SUBAPPLICATION Uebung_230 (* Analog-Eingang *)
  (* Standard: 61499-2; Description: Copyright (c) 2023 Meisterschulen am Ostbahnhof This program and the accompanying materials are made available under the terms of the Eclipse Public License 2.0 which is available at https://www.eclipse.org/legal/epl-2.0/ SPDX-License-Identifier: EPL-2.0 *)
  (* Version 1.0, 2023-10-23, Franz Höpfinger, Meisterschulen am Ostbahnhof, initial API and implementation and/or initial documentation *)
  PACKAGE Uebungen;
  IMPORT DataPanel::io::MI::AI::DataPanel_MI_AI::AnalogInput_1A;
  IMPORT DataPanel::io::MI::const::MI::MI_00;
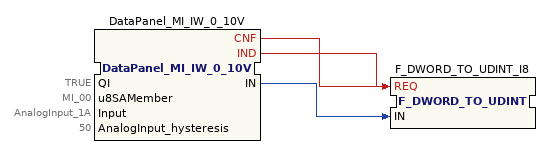
  FBS
    DataPanel_MI_IW_0_10V : DataPanel::io::MI::AI::DataPanel_MI_IW_0_10V(QI := TRUE, u8SAMember := MI_00, Input := AnalogInput_1A, AnalogInput_hysteresis := 50);
    F_DWORD_TO_UDINT_I8 : iec61131::conversion::F_DWORD_TO_UDINT;
  END_FBS
  EVENT_CONNECTIONS
    DataPanel_MI_IW_0_10V.CNF TO F_DWORD_TO_UDINT_I8.REQ;
    DataPanel_MI_IW_0_10V.IND TO F_DWORD_TO_UDINT_I8.REQ;
  END_CONNECTIONS
  DATA_CONNECTIONS
    DataPanel_MI_IW_0_10V.IN TO F_DWORD_TO_UDINT_I8.IN;
  END_CONNECTIONS
END_SUBAPPLICATION
